{attribute 'GeneratedUsingTerminal: EP7211-0035-0029'}
{attribute addProperty BoxType "EP7211-0035-0029"}
{attribute addProperty Id "Position_actual_valueAT %I*UDINT4"}
{attribute addProperty CRC "131878004"}
{attribute addProperty Size "4"}
TYPE DS402_Position_actual_value_07DC4C74 :
STRUCT
	{attribute addProperty Name "Position_actual_value"}
	Position_actual_value AT %I* : UDINT;
END_STRUCT
END_TYPE

(* stored: Version 1.2.0.0, ProductVersion 3.1.4024.9
   DUT DS402_Position_actual_value_07DC4C74: Id {aef0b6da-2e29-4535-aeaf-adad4045d34e} *)
